(* IEC 61131-3 sources: Berechnungsplattform/PLC_CODESYS, 2 files *)

(* ---- GVL_Joystick.st ---- *)
(* ============================================================================
   Global Variable List: GVL_Joystick
   Development Environment: CODESYS
   PLC Hardware: Intercontrol DIGSY Fusion S
   Description: Global variables for joystick and CAN communication system
   ============================================================================ *)
{attribute 'qualified_only'}
VAR_GLOBAL
    (* CAN Configuration *)
    CAN_BAUDRATE        : DWORD := 250000;      (* CAN Baudrate in bit/s *)
    JOYSTICK_BASE_ID    : DWORD := 16#180;      (* Base CAN ID for Gessmann joystick *)
    THRUST_LEVER_ID     : DWORD := 16#181;      (* CAN ID for thrust lever *)
    BUTTONS_ID          : DWORD := 16#182;      (* CAN ID for buttons *)
    COMM_TIMEOUT        : TIME := T#500MS;      (* Communication timeout *)
    CYCLE_TIME          : TIME := T#10MS;       (* PLC cycle time *)

    (* Deadzone settings in percent *)
    DEADZONE_X          : REAL := 5.0;          (* Deadzone for X-axis *)
    DEADZONE_Y          : REAL := 5.0;          (* Deadzone for Y-axis *)
    DEADZONE_Z          : REAL := 5.0;          (* Deadzone for Z-axis/rotation *)
    DEADZONE_THRUST     : REAL := 2.0;          (* Deadzone for thrust lever *)

    (* Thrust limits and rates *)
    MAX_THRUST          : REAL := 100.0;        (* Maximum thrust limit (%) *)
    MIN_THRUST          : REAL := -30.0;        (* Minimum thrust limit (%) *)
    RAMP_UP_RATE        : REAL := 50.0;         (* Acceleration rate (%/s) *)
    RAMP_DOWN_RATE      : REAL := 75.0;         (* Deceleration rate (%/s) *)
    EMERGENCY_RAMP_RATE : REAL := 200.0;        (* Emergency stop rate (%/s) *)
    DEADBAND            : REAL := 2.0;          (* Input deadband (%) *)

    (* System status flags - read/write from other programs *)
    System_Ready        : BOOL := FALSE;        (* System is ready for operation *)
    Emergency_Active    : BOOL := FALSE;        (* Emergency stop is active *)
    CAN_Online          : BOOL := FALSE;        (* CAN communication is online *)
    Joystick_Online     : BOOL := FALSE;        (* Joystick is communicating *)

    (* Error codes *)
    System_Error_Code   : DWORD := 0;           (* Current system error code *)
    (* Error code definitions:
       0 = No error
       1 = CAN not initialized
       2 = Joystick offline/timeout
       3 = Joystick communication error
       4 = Emergency stop active
    *)
END_VAR

(* ---- Main_Control.st ---- *)
(* ============================================================================
   Main Control Program
   Development Environment: CODESYS
   PLC Hardware: Intercontrol DIGSY Fusion S
   Description: Main control program integrating CAN communication,
                Gessmann joystick, and thrust lever control
   ============================================================================ *)

PROGRAM PLC_PRG
VAR
    (* CAN Interface *)
    fbCANInterface      : FB_CAN_Interface;
    bCANEnable          : BOOL := TRUE;
    dwCANBaudrate       : DWORD := 250000;      (* 250 kbit/s standard for Gessmann *)

    (* Joystick Handler *)
    fbJoystick          : FB_Gessmann_Joystick;
    bJoystickEnable     : BOOL := TRUE;
    dwJoystickBaseID    : DWORD := 16#180;      (* Base CAN ID for Gessmann joystick *)

    (* Thrust Lever Control *)
    fbThrustControl     : FB_Thrust_Lever_Control;
    bThrustEnable       : BOOL := TRUE;
    eThrustMode         : Thrust_Mode := THRUST_MODE_RAMP;

    (* Control outputs *)
    rDriveSpeedX        : REAL := 0.0;          (* X-axis drive speed command *)
    rDriveSpeedY        : REAL := 0.0;          (* Y-axis drive speed command *)
    rRotationSpeed      : REAL := 0.0;          (* Rotation speed command *)
    rThrustCommand      : REAL := 0.0;          (* Thrust command *)

    (* Status and diagnostics *)
    bSystemReady        : BOOL := FALSE;
    bCANOnline          : BOOL := FALSE;
    bJoystickOnline     : BOOL := FALSE;
    bThrustActive       : BOOL := FALSE;
    dwErrorCode         : DWORD := 0;

    (* Safety *)
    bEmergencyStop      : BOOL := FALSE;
    bSafetyOK           : BOOL := TRUE;

    (* Timing *)
    tCycleTime          : TIME := T#10MS;
END_VAR

(* ============================================================================
   Main Control Logic
   ============================================================================ *)

(* Initialize CAN Interface *)
fbCANInterface(
    bEnable := bCANEnable,
    dwBaudrate := dwCANBaudrate
);

bCANOnline := fbCANInterface.bInitialized;

(* Process Joystick *)
fbJoystick(
    bEnable := bJoystickEnable AND bCANOnline,
    stCANMessage := fbCANInterface.stRxMessage,
    bNewCANMessage := fbCANInterface.bMessageReceived,
    dwJoystickCANID := dwJoystickBaseID,
    dwThrustLeverCANID := dwJoystickBaseID + 1,
    dwButtonsCANID := dwJoystickBaseID + 2,
    tTimeout := T#500MS,
    rDeadzoneX := 5.0,
    rDeadzoneY := 5.0,
    rDeadzoneZ := 5.0,
    rDeadzoneThrustLever := 2.0
);

bJoystickOnline := fbJoystick.bOnline;

(* Process Thrust Lever Control *)
fbThrustControl(
    bEnable := bThrustEnable AND bJoystickOnline AND bSafetyOK,
    rThrustLeverInput := fbJoystick.rThrustLever,
    eRequestedMode := eThrustMode,
    bEmergencyStop := bEmergencyStop,
    bCruiseSet := fbJoystick.stJoystickData.bButton1,
    bCruiseResume := fbJoystick.stJoystickData.bButton2,
    bCruiseCancel := fbJoystick.stJoystickData.bButton3,
    rMaxThrust := 100.0,
    rMinThrust := -30.0,    (* Limit reverse thrust *)
    rRampUpRate := 50.0,
    rRampDownRate := 75.0,
    rEmergencyRampRate := 200.0,
    rDeadband := 2.0,
    tCycleTime := tCycleTime
);

bThrustActive := fbThrustControl.bActive;

(* Map joystick outputs to control commands *)
IF bSafetyOK AND NOT bEmergencyStop THEN
    (* Normal operation *)
    rDriveSpeedX := fbJoystick.rAxisX;
    rDriveSpeedY := fbJoystick.rAxisY;
    rRotationSpeed := fbJoystick.rAxisZ;
    rThrustCommand := fbThrustControl.rThrustOutput;
ELSE
    (* Safe state - all outputs to zero *)
    rDriveSpeedX := 0.0;
    rDriveSpeedY := 0.0;
    rRotationSpeed := 0.0;
    rThrustCommand := 0.0;
END_IF

(* System ready status *)
bSystemReady := bCANOnline AND bJoystickOnline AND bSafetyOK AND NOT bEmergencyStop;

(* Error handling *)
IF NOT bCANOnline THEN
    dwErrorCode := 1;   (* CAN not initialized *)
ELSIF NOT bJoystickOnline THEN
    dwErrorCode := 2;   (* Joystick offline *)
ELSIF fbJoystick.bError THEN
    dwErrorCode := 3;   (* Joystick error *)
ELSIF fbThrustControl.stStatus.bEmergency THEN
    dwErrorCode := 4;   (* Emergency stop active *)
ELSE
    dwErrorCode := 0;   (* No error *)
END_IF

(* Update global status variables *)
GVL_Joystick.System_Ready := bSystemReady;
GVL_Joystick.Emergency_Active := bEmergencyStop;
GVL_Joystick.CAN_Online := bCANOnline;
GVL_Joystick.Joystick_Online := bJoystickOnline;
GVL_Joystick.System_Error_Code := dwErrorCode;

END_PROGRAM
